Omron CX-Programmer project NewProject (CX-Programmer 9.75)

# PLC NewPLC1: CP1L M

## Global symbols (name address type ; comment)
0.00 BOOL  ; X0
0.01 BOOL  ; X1
100.00 BOOL  ; Y0
100.01 BOOL  ; Y1

## Program NewProgram1 (cyclic task 0)

### Section Section1

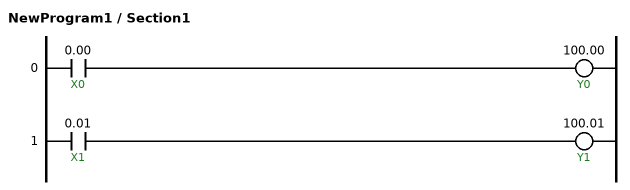
; rung 0
LD 0.00  ; X0
OUT 100.00  ; Y0
; rung 1
LD 0.01  ; X1
OUT 100.01  ; Y1

### Section END
; rung 0
END(001)